(*******************************************************************************
                          protoc-gen-twincat V0.0.0.0                           
                  https://github.com/TcHaxx/protoc-gen-twincat                  
*******************************************************************************)
{attribute 'no_explicit_call' := 'do not call this POU directly'}
{attribute 'no-analysis'}
// Another message demonstrating all field options
FUNCTION_BLOCK INTERNAL FINAL FB_ComplexData IMPLEMENTS I_Message
VAR
    _fbMessageParser : FB_MessageParser(ipMessage:= THIS^);
    _fbMessageWriter : FB_MessageWriter(ipMessage:= THIS^);
    _stComplexData : ST_ComplexData;
    // repeated uint32 array_data = 5;
    _fbFieldCodecId5 : FB_FieldCodecUint32(nTag:= 16#2A);
    _fbRepeatedId5 : FB_RepeatedField(anyArray:= F_ToAnyType(_stComplexData.array_data), anyFirstElem:= F_ToAnyType(_stComplexData.array_data[0]), ipFieldCodec:= _fbFieldCodecId5);
    // repeated SensorReading readings = 10;
    _fbFieldCodecId10 : FB_FieldCodecMessage(nTag:= 16#52, ipMessage:= _fbreadings);
    _fbRepeatedId10 : FB_RepeatedField(anyArray:= F_ToAnyType(_stComplexData.readings), anyFirstElem:= F_ToAnyType(_stComplexData.readings[0]), ipFieldCodec:= _fbFieldCodecId10);
    _fbreadings : FB_SensorReading;
    END_VAR

{attribute 'no-analysis'}
(* Calculates the size of this message in Protocol Buffer wire format, in bytes. *)
METHOD CalculateSize : UDINT
VAR
    nSize : UDINT;
    nRepeatedFieldSize : UDINT;
END_VAR
// string label = 1;
nSize := nSize + 1 + F_ComputeStringSize(anyString:= _stComplexData.label);
// int32 value_dint = 2;
nSize := nSize + 1 + F_ComputeInt32Size(anyDint:= _stComplexData.value_dint);
// int32 value_int = 3;
nSize := nSize + 1 + F_ComputeInt32Size(anyDint:= _stComplexData.value_int);
// uint32 value_word = 4;
nSize := nSize + 1 + F_ComputeUint32Size(anyUdint:= _stComplexData.value_word);
// repeated uint32 array_data = 5;
_fbRepeatedId5.nCount := _stComplexData.array_data_count;
_fbRepeatedId5.CalculateSize(nSize => nRepeatedFieldSize);
nSize := nSize + nRepeatedFieldSize;
// Status state = 6;
nSize := nSize + 1 + F_ComputeEnumSize(anyEnum:= _stComplexData.state);
// bytes raw_bytes = 7;
nSize := nSize + 1 + F_ComputeBytesSize(aBytes:= _stComplexData.raw_bytes, nCount:= _stComplexData.raw_bytes_count);
// double measurement = 8;
nSize := nSize + 1 + F_ComputeDoubleSize(fValue:= _stComplexData.measurement);
// float calibration_factor = 9;
nSize := nSize + 1 + F_ComputeFloatSize(fValue:= _stComplexData.calibration_factor);
// repeated SensorReading readings = 10;
_fbRepeatedId10.nCount := _stComplexData.readings_count;
_fbRepeatedId10.CalculateSize(nSize => nRepeatedFieldSize);
nSize := nSize + nRepeatedFieldSize;
// DataType data_type = 11;
nSize := nSize + 1 + F_ComputeEnumSize(anyEnum:= _stComplexData.data_type);
CalculateSize := nSize;
END_METHOD

PROPERTY PUBLIC ComplexData : ST_ComplexData
GET
ComplexData := _stComplexData;
END_GET
SET
_stComplexData := ComplexData;
// repeated SensorReading readings = 10;
_stComplexData.readings := ComplexData.readings;
END_SET
END_PROPERTY

(* Merges the data from the specified coded input stream with the current message.*)
{attribute 'no-analysis'}
METHOD MergeFrom : HRESULT
VAR_IN_OUT
    fbParseCtx : FB_ParseContext;
END_VAR
VAR
    nTag : UDINT;
END_VAR
_fbRepeatedId10.Initialize();
_fbRepeatedId5.Initialize();
REPEAT
MergeFrom := fbParseCtx.ReadTag(nTag=> nTag);
IF SUCCEEDED(MergeFrom) AND nTag = 0 THEN
    EXIT;
END_IF;

IF FAILED(MergeFrom) THEN
    RETURN;
END_IF

CASE nTag OF
    16#0A:    // string label = 1;
        MergeFrom := fbParseCtx.ReadString(anyStringOut:= _stComplexData.label); 
    16#10:    // int32 value_dint = 2;
        MergeFrom := fbParseCtx.ReadInt32(anyDint:= _stComplexData.value_dint); 
    16#18:    // int32 value_int = 3;
        MergeFrom := fbParseCtx.ReadInt32(anyDint:= _stComplexData.value_int); 
    16#20:    // uint32 value_word = 4;
        MergeFrom := fbParseCtx.ReadUint32(anyUdint:= _stComplexData.value_word); 
    16#2A:    // repeated uint32 array_data = 5;
        MergeFrom := _fbRepeatedId5.AddEntriesFrom(fbParseCtx:= fbParseCtx, ipFieldCodec:= _fbFieldCodecId5,nCount=> _stComplexData.array_data_count);
    16#30:    // Status state = 6;
        MergeFrom := fbParseCtx.ReadEnum(anyEnum:= _stComplexData.state); 
    16#3A:    // bytes raw_bytes = 7;
        MergeFrom := fbParseCtx.ReadBytes(aBytes:= _stComplexData.raw_bytes, nCount=> _stComplexData.raw_bytes_count); 
    16#41:    // double measurement = 8;
        MergeFrom := fbParseCtx.ReadDouble(fValue=> _stComplexData.measurement); 
    16#4D:    // float calibration_factor = 9;
        MergeFrom := fbParseCtx.ReadFloat(fValue=> _stComplexData.calibration_factor); 
    16#52:    // repeated SensorReading readings = 10;
        MergeFrom := _fbRepeatedId10.AddEntriesFrom(fbParseCtx:= fbParseCtx, ipFieldCodec:= _fbFieldCodecId10,nCount=> _stComplexData.readings_count);
    16#58:    // DataType data_type = 11;
        MergeFrom := fbParseCtx.ReadEnum(anyEnum:= _stComplexData.data_type); 
ELSE
    MergeFrom := fbParseCtx.SkipLastField();
END_CASE

UNTIL (FAILED(MergeFrom) OR nTag = 0)
END_REPEAT
END_METHOD

PROPERTY PUBLIC MessageValue : T_Any
GET
MessageValue := F_ToAnyType(anyArg:= _stComplexData);
END_GET
END_PROPERTY

PROPERTY PUBLIC Parser : REFERENCE TO FB_MessageParser
GET
Parser REF= THIS^._fbMessageParser;
END_GET
END_PROPERTY

(* Writer for this message.*)
PROPERTY PUBLIC Writer : REFERENCE TO FB_MessageWriter
GET
Writer REF= THIS^._fbMessageWriter;
END_GET
END_PROPERTY

(* Writes the data to the given coded output stream.*)
{attribute 'no-analysis'}
METHOD WriteTo : HRESULT
VAR_IN_OUT
	(* Coded output stream to write the data to. *)
	fbWriteCtx	: FB_WriteContext;
END_VAR
// string label = 1;
WriteTo := fbWriteCtx.WriteTag(1, E_WireType.LengthDelimited);
IF FAILED(WriteTo) THEN
    RETURN;
END_IF
WriteTo := fbWriteCtx.WriteString(sStringToWrite:= _stComplexData.label);
IF FAILED(WriteTo) THEN
    RETURN;
END_IF
// int32 value_dint = 2;
WriteTo := fbWriteCtx.WriteTag(2, E_WireType.Varint);
IF FAILED(WriteTo) THEN
    RETURN;
END_IF
WriteTo := fbWriteCtx.WriteInt32(anyDint:= _stComplexData.value_dint);
IF FAILED(WriteTo) THEN
    RETURN;
END_IF
// int32 value_int = 3;
WriteTo := fbWriteCtx.WriteTag(3, E_WireType.Varint);
IF FAILED(WriteTo) THEN
    RETURN;
END_IF
WriteTo := fbWriteCtx.WriteInt32(anyDint:= _stComplexData.value_int);
IF FAILED(WriteTo) THEN
    RETURN;
END_IF
// uint32 value_word = 4;
WriteTo := fbWriteCtx.WriteTag(4, E_WireType.Varint);
IF FAILED(WriteTo) THEN
    RETURN;
END_IF
WriteTo := fbWriteCtx.WriteUint32(anyUdint:= _stComplexData.value_word);
IF FAILED(WriteTo) THEN
    RETURN;
END_IF
// repeated uint32 array_data = 5;
WriteTo := _fbRepeatedId5.WriteToWithCount(fbWriteCtx:= fbWriteCtx, ipFieldCodec:= _fbFieldCodecId5, nCount:= _stComplexData.array_data_count);
IF FAILED(WriteTo) THEN
    RETURN;
END_IF
// Status state = 6;
WriteTo := fbWriteCtx.WriteTag(6, E_WireType.Varint);
IF FAILED(WriteTo) THEN
    RETURN;
END_IF
WriteTo := fbWriteCtx.WriteEnum(anyEnum:= _stComplexData.state);
IF FAILED(WriteTo) THEN
    RETURN;
END_IF
// bytes raw_bytes = 7;
WriteTo := fbWriteCtx.WriteTag(7, E_WireType.LengthDelimited);
IF FAILED(WriteTo) THEN
    RETURN;
END_IF
WriteTo := fbWriteCtx.WriteBytes(aBytes:= _stComplexData.raw_bytes, nCount:= _stComplexData.raw_bytes_count);
IF FAILED(WriteTo) THEN
    RETURN;
END_IF
// double measurement = 8;
WriteTo := fbWriteCtx.WriteTag(8, E_WireType.Fixed64);
IF FAILED(WriteTo) THEN
    RETURN;
END_IF
WriteTo := fbWriteCtx.WriteDouble(fValue:= _stComplexData.measurement);
IF FAILED(WriteTo) THEN
    RETURN;
END_IF
// float calibration_factor = 9;
WriteTo := fbWriteCtx.WriteTag(9, E_WireType.Fixed32);
IF FAILED(WriteTo) THEN
    RETURN;
END_IF
WriteTo := fbWriteCtx.WriteFloat(fValue:= _stComplexData.calibration_factor);
IF FAILED(WriteTo) THEN
    RETURN;
END_IF
// repeated SensorReading readings = 10;
WriteTo := _fbRepeatedId10.WriteToWithCount(fbWriteCtx:= fbWriteCtx, ipFieldCodec:= _fbFieldCodecId10, nCount:= _stComplexData.readings_count);
IF FAILED(WriteTo) THEN
    RETURN;
END_IF
// DataType data_type = 11;
WriteTo := fbWriteCtx.WriteTag(11, E_WireType.Varint);
IF FAILED(WriteTo) THEN
    RETURN;
END_IF
WriteTo := fbWriteCtx.WriteEnum(anyEnum:= _stComplexData.data_type);
IF FAILED(WriteTo) THEN
    RETURN;
END_IF
END_METHOD

END_FUNCTION_BLOCK

(* stored: Version 1.1.0.1
   POU FB_ComplexData: Id {a8c3f68e-aac3-4a2a-a70e-41bd6566c60b}, SpecialFunc None
   Method CalculateSize: Id {3f3f837a-5da0-437b-ab54-d10045771ac5}
   Property ComplexData: Id {8af5940d-bd13-469f-96e2-28ee6a0aabd3}
   Get Get: Id {2b7e1d5b-7c4d-4742-b0cc-c01d1d58c8f8}
   Set Set: Id {7c625bc7-d49b-4d2f-b583-da62edf5d656}
   Method MergeFrom: Id {6ba37205-228b-4cc0-8e94-ca71847f98d2}
   Property MessageValue: Id {4cef794e-8c13-40f2-9a08-cc70dd76bcd8}
   Get Get: Id {65fec3f4-5fb3-4ce9-a6ab-ef6d0d770d25}
   Property Parser: Id {082b6dce-4600-4e1d-8364-7603b8c9b7c7}
   Get Get: Id {fd39de4e-451e-4471-9fc2-9daa69ddfd85}
   Property Writer: Id {f4b7af37-7162-4565-aead-dc0cdad3ccf4}
   Get Get: Id {28281246-9964-4582-b6d7-a51d3d262fe3}
   Method WriteTo: Id {7e68a930-43de-46c2-8559-305dc4282d7e} *)
